VAR_GLOBAL // STATE
    inp: LREAL;
    c: LREAL;
    aut_r: LREAL;
    aut_b: BOOL;
    aut_i: DINT;
    aut_tii: TupleStruct;
    aut_i2: DINT;
    aut_i3: DINT;
    aut: aut_location;
END_VAR

(* stored: ProductVersion 3.1.0.18, Version 1.1.0.1 *)
